Fanuc KAREL source: UNLOCK_GROUP.kl

PROGRAM T
%NOLOCKGROUP
VAR
 v0 : INTEGER
 v1 : INTEGER
BEGIN
 UNLOCK_GROUP(v0, v1)
END T
